SUBAPPLICATION Uebung_236_AX (* AX_LAST_2: derselbe Last-Wins-auf-jeder-Flanke-Effekt wie Uebung_229/230/233_AX, aber ohne Edge-Detektor+Latch - Q1 folgt direkt dem zuletzt geschriebenen AX-Socket *)
  (* Standard: 61499-2; Description: Copyright (c) 2026 Meisterschulen am Ostbahnhof This program and the accompanying materials are made available under the terms of the Eclipse Public License 2.0 which is available at https://www.eclipse.org/legal/epl-2.0/ SPDX-License-Identifier: EPL-2.0 *)
  (* Version 1.0, 2026-09-07, Franz Höpfinger, Meisterschulen am Ostbahnhof, initial API and implementation and/or initial documentation *)
  PACKAGE Uebungen;
  IMPORT logiBUS::io::DI::logiBUS_DI::Input_I1;
  IMPORT logiBUS::io::DI::logiBUS_DI::Input_I2;
  IMPORT logiBUS::io::DQ::logiBUS_DO::Output_Q1;
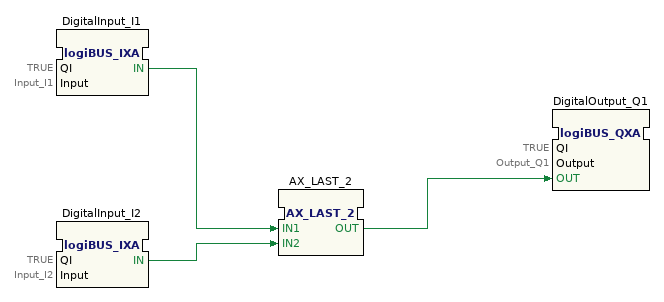
  FBS
    DigitalInput_I1 : logiBUS::io::DI::logiBUS_IXA(QI := TRUE, Input := Input_I1);
    DigitalInput_I2 : logiBUS::io::DI::logiBUS_IXA(QI := TRUE, Input := Input_I2);
    AX_LAST_2 : adapter::events::unidirectional::AX_LAST_2;
    DigitalOutput_Q1 : logiBUS::io::DQ::logiBUS_QXA(QI := TRUE, Output := Output_Q1);
  END_FBS
  ADAPTER_CONNECTIONS
    DigitalInput_I1.IN TO AX_LAST_2.IN1;
    DigitalInput_I2.IN TO AX_LAST_2.IN2;
    AX_LAST_2.OUT TO DigitalOutput_Q1.OUT;
  END_CONNECTIONS
END_SUBAPPLICATION
